// TIA Portal V20 export
FUNCTION_BLOCK "Simulation"   // FB50097, LAD
// stored: MemoryReserve 100, Namespace Unit1.Em3, SetENOAutomatically false
   VAR_INPUT
      simulation { ExternalAccessible := 'False'; ExternalVisible := 'False'; ExternalWritable := 'False'} : Bool;
   END_VAR
   VAR
      instActuator { ExternalAccessible := 'False'; ExternalVisible := 'False'; ExternalWritable := 'False'} : Array[0..19] of "LER_SimActuator";
   END_VAR
BEGIN

REGION Network 1: Two Way Actuator
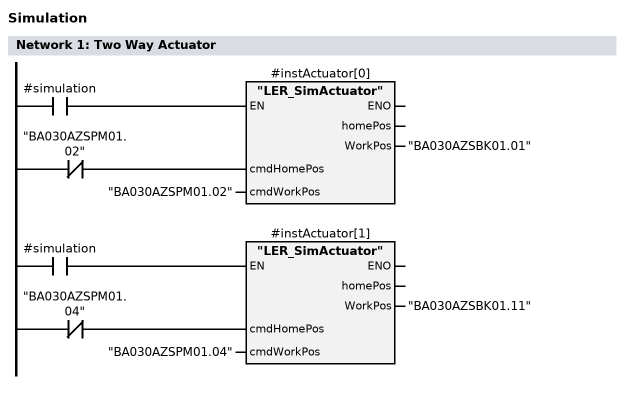
   RUNG wire#powerrail
      Contact( #simulation )
      #instActuator[0](cmdHomePos := wire#w1, cmdWorkPos := "BA030AZSPM01.02", homePos =>, WorkPos => "BA030AZSBK01.01")
   END_RUNG
   RUNG wire#powerrail
      I_Contact( "BA030AZSPM01.02" )
   END_RUNG wire#w1
   RUNG wire#powerrail
      Contact( #simulation )
      #instActuator[1](cmdHomePos := wire#w2, cmdWorkPos := "BA030AZSPM01.04", homePos =>, WorkPos => "BA030AZSBK01.11")
   END_RUNG
   RUNG wire#powerrail
      I_Contact( "BA030AZSPM01.04" )
   END_RUNG wire#w2
   // the same network as SCL:
   IF #simulation THEN
       #instActuator[0](cmdHomePos := NOT "BA030AZSPM01.02",   // "LER_SimActuator"
                        cmdWorkPos := "BA030AZSPM01.02",
                        WorkPos => "BA030AZSBK01.01");
       #instActuator[1](cmdHomePos := NOT "BA030AZSPM01.04",   // "LER_SimActuator"
                        cmdWorkPos := "BA030AZSPM01.04",
                        WorkPos => "BA030AZSBK01.11");
   END_IF;
END_REGION
END_FUNCTION_BLOCK
